FUNCTION_BLOCK SludgeBufferSensors_HMI (* Service Interface Function Block Type *)
  (* Standard: 61499-2 *)
  (* Version 0.0, 7/1/2024, NVPP, Schneider Electric, template *)
  PACKAGE SE.Nereda;
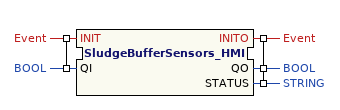
  EVENT_INPUT
    INIT WITH QI;
  END_EVENT
  EVENT_OUTPUT
    INITO WITH QO, STATUS;
  END_EVENT
  VAR_INPUT
    QI : BOOL;
  END_VAR
  VAR_OUTPUT
    QO : BOOL; (* Event Output Qualifier *)
    STATUS : STRING; (* Service Status *)
  END_VAR
  SERVICE /
    SEQUENCE 
    END_SEQUENCE
  END_SERVICE
END_FUNCTION_BLOCK
